TYPE ST_OpenLoopControlWinchSettings :
STRUCT
	fWichDrumDiameter : LREAL := 0.0475;
	fWinchDisplacement : LREAL := 32;
	fGearBox : LREAL := 20;
	fMaxFlow : LREAL := 60;
	fWinchDrumScaling : LREAL := 0.000744309;
END_STRUCT
END_TYPE

(* stored: Version 1.1.0.1, ProductVersion 3.1.4024.12
   DUT ST_OpenLoopControlWinchSettings: Id {a3f73810-9df0-4ca0-9bf3-dd6dbbdd159d} *)
